FUNCTION_BLOCK FB_Doubly_Linked_List IMPLEMENTS I_Linked_List
VAR
	pHead :  POINTER TO ST_NODE;
	pTail :  POINTER TO ST_NODE;
	t_Null: T_DATA_TYPE;
END_VAR

(* Creates/Adds an node to the end of the list. *)
METHOD Create
VAR_INPUT
	(* Data to add to new node.*)
	Data		: T_DATA_TYPE;
END_VAR
VAR
	pTemp 		:  POINTER TO ST_NODE; //  New node will be allocated at this pointer
	pPrevious 	: POINTER TO ST_NODE; // Previous node location will be stored at this pointer temporarily
END_VAR
pTemp := __NEW(ST_NODE);
pTemp^.Data := Data;
IF THIS^.pHead = 0 THEN 
	THIS^.pHead := pTemp; 
	THIS^.pTail := THIS^.pHead; // If the pointer to the pHead is NULL then give it an address. The pTail address of the first node is the pHead.
ELSE
	pPrevious := THIS^.pTail;
	THIS^.pTail^.pNext := pTemp; 
	THIS^.pTail := pTemp;
	THIS^.pTail^.pPrevious := pPrevious; 
	END_IF // Point previous node's pNext to the address of pTemp and set pTail to pTemp.
END_METHOD

(* Empties/Clears/Deletes list*)
METHOD Empty
VAR
	pTemp : POINTER TO ST_NODE;
END_VAR
pTail := 0;
pTemp := pHead;
WHILE pTemp <> 0 DO
	pTemp := pTemp^.pNext; THIS^.Pop();
END_WHILE
END_METHOD

METHOD FB_exit : BOOL
VAR_INPUT
	(* if TRUE, the exit method is called for exiting an instance that is copied afterwards (online change).*)
	bInCopyCode	: BOOL;
END_VAR
This^.Empty();
END_METHOD

METHOD FB_init : BOOL
VAR_INPUT
	(* if TRUE, the retain variables are initialized (warm start / cold start)*)
	bInitRetains	: BOOL;
	(* if TRUE, the instance afterwards gets moved into the copy code (online change)*)
	bInCopyCode	: BOOL;
END_VAR
END_METHOD

(* Inserts node at a specific position in the list*)
METHOD Insert
VAR_INPUT
	(* Data to add to new node.*)
	Data	: T_DATA_TYPE;
	(* Position to add new node in list.*)
	nPosition	: DINT;
END_VAR
END_METHOD

(* Checks of list is empty.*)
METHOD Is_Empty : BOOL
END_METHOD

(* Gets element at any position of the list, wuthout removing it.*)
METHOD Peek : T_DATA_TYPE
VAR_INPUT
	nPosition	: DINT;
END_VAR
END_METHOD

(* Deletes/pops a node at the front of the list *)
METHOD Pop : T_DATA_TYPE
VAR
	pTemp : POINTER TO ST_NODE;
END_VAR
IF THIS^.pHead = 0 THEN RETURN; END_IF 
Pop := pHead^.Data;
pTemp := pHead^.pNext;
__DELETE(pHead);
pHead := pTemp;
END_METHOD

(* Adds/pushes a node at the front of the list *)
METHOD Push
VAR_INPUT
	Data	: T_DATA_TYPE;
END_VAR
END_METHOD

(* Deletes node at a specific position in the list*)
METHOD Remove : T_DATA_TYPE
VAR_INPUT
	(* Position of node to delete.*)
	nPosition	: DINT;
END_VAR
END_METHOD

(* Reverse list*)
METHOD Reverse
END_METHOD

//{warning 'add method implementation '}
(* Searches list for the first instance of data and returns it's location and whether it's in the list.*)
METHOD Search : BOOL
VAR_INPUT
	(* Data to find in list*)
	Data	: T_DATA_TYPE;
END_VAR
VAR_OUTPUT
	(* Location of the data  starting from 1. 0 means data is not found in list*)
	nPosition	: DINT;
END_VAR
END_METHOD

(* Traverse the list to display each node. *)
METHOD Show
VAR_IN_OUT
	aList 		: ARRAY[*] OF T_DATA_TYPE; // Array to display data in list.
END_VAR
VAR
	pCurrent 	: POINTER TO ST_NODE;
	i 			: DINT;
END_VAR
END_METHOD

(* Gets size of the list*)
METHOD Size : DINT
END_METHOD

END_FUNCTION_BLOCK

(* stored: Version 1.1.0.1, ProductVersion 3.1.4024.4
   POU FB_Doubly_Linked_List: Id {03f6cb54-b49e-4d08-867b-b49ddd590b59}, SpecialFunc None
   Method Create: Id {6e81400d-b895-4d17-b1a0-7da2503c1458}
   Method Empty: Id {13f871b3-e858-4291-a8b3-2f75777917f4}
   Method FB_exit: Id {941d640c-d7b3-4d27-8004-bad3bfec5e67}
   Method FB_init: Id {068ef67d-337f-4431-90f7-195c921196d4}
   Method Insert: Id {a2deca27-6648-4030-8273-4c1592694cd7}
   Method Is_Empty: Id {7916821b-b988-42e5-9364-676420ec6aa8}
   Method Peek: Id {1abc0c76-03e0-4d2b-aeef-61f5be63a525}
   Method Pop: Id {9494d023-f6c0-4f2d-a8f8-1220fb5899b4}
   Method Push: Id {df0359e8-209b-4c98-944c-e2caa380bbd6}
   Method Remove: Id {6e058adb-4972-4a7b-a117-85ef4a2c1908}
   Method Reverse: Id {62dd27d4-3e49-4101-aef8-53ee263ebe87}
   Method Search: Id {c1b15b75-1452-4c17-83dd-a4eb41b967d7}
   Method Show: Id {38cfe029-c78d-4d3d-a50d-75c428b2b275}
   Method Size: Id {3a7822bb-5a82-43d8-9eae-6b968a22a256} *)
